Staubli VAL3: TCPserver.pgx

program TCPserver()
  local num l_nStatus
  local num l_nBytesIn[24]
  local num l_nSuccBytes
begin
  // l_nBytesIn: 24 bit -> 3 byte
  // nData: 3
  while true
    logMsg("Schleife start")
    l_nStatus=sioGet(soTcpClient, l_nBytesIn)
    if l_nStatus>0
      // Write recieved bytes in data
      // Achtung bei mehr Bitlänge 24, 3 und globale Variable(nData) ändern
      logMsg("Empfangene Daten sind fehlerhaft",2)
      if(fromBinary(l_nBytesIn,24,"8.0l",nData)!=3)
      else
        logMsg("Daten über TCP/IP empfangen")
        // check if data is in limits
        // ...
        nX = limit(nData[0],1,4)
        nY = limit(nData[1],1,3)
        if nData[2]>0
          bPick = true
        else
          bPick = false
        endIf
        bReady = false
        bNewData = true
      endIf

      // tell client that robot is ready
      wait(bReady)

      //delay(2)
      l_nStatus=sioSet(soTcpClient, 1)
    endIf
  endWhile
end
